{attribute addProperty BoxType "EL3773-0000-0018"}
{attribute addProperty Id "StartTimeNextLatchAT %I*StartTimeNextLatch_356BEDAC648"}
{attribute addProperty CRC "1421024673"}
{attribute addProperty SizeInBites "64"}
{attribute addProperty SizeInBytes "8"}
TYPE AI_NextSync1Time_54B31DA1 :
STRUCT
	{attribute addProperty Name "StartTimeNextLatch"}
	StartTimeNextLatch AT %I* : StartTimeNextLatch_356BEDAC;
END_STRUCT
END_TYPE

(* stored: Version 1.2.0.0, ProductVersion 3.1.4024.9
   DUT AI_NextSync1Time_54B31DA1: Id {e0d8e9e7-7cce-4b1c-b001-a994dfee69c0} *)
